// TIA Portal V21 export
DATA_BLOCK "DB603"   // DB603
TITLE = DB603
AUTHOR : PRECISE
FAMILY : PRECISE
// CycleSelection
// stored: AutoNumber false, InstanceOfName FB603, InstanceOfType FB
"FB603"
   // VAR_INPUT
   //    CycleEnable : Bool;
   //    CycleRunning : Bool;
   //    SecPulse : Bool;
   //    AlwaysTrue : Bool;
   //    CycleSelection : "CIP";
   //    ConductivitySuccessWhileRinse : Bool;
   //    ConductivitySuccessWhileDrain : Bool;
   //    ConductivitySuccessWhileTransfer : Bool;
   // END_VAR
   // VAR_OUTPUT
   //    Started : Bool;
   //    VentValve : Bool;
   //    PrintActualRep : Int;
   // END_VAR
   // VAR_IN_OUT
   //    Over : Bool;
   //    OverTemp : Bool;
   //    RepeatCycle : Bool;
   //    ActualRepetition : Int;
   //    CycleStart : "CipCycleStarted";
   //    CycleOver : "CipCycleOver";
   //    ConductivityStatus : Bool;
   //    TimeSaveModeRep : Int;
   //    StartFillingToSaveTime : Bool;
   //    Reset : Bool;
   //    RecirculationPopupTemp : Bool;
   //    RecirculationPopupTempAck : Bool;
   // END_VAR
   // VAR
   //    Re : Array[0..30] of Bool;
   // END_VAR
BEGIN
END_DATA_BLOCK
